(* CODESYS project proldPlcPrg.export

Project tree, tasks and I/O mapping:
  program PLC_PRG [LD]
*)

// PLC_PRG
PROGRAM PLC_PRG
VAR
	tmPusher1: TP;
	tmPusher2: TP;
	tmPusher3: TP;
END_VAR

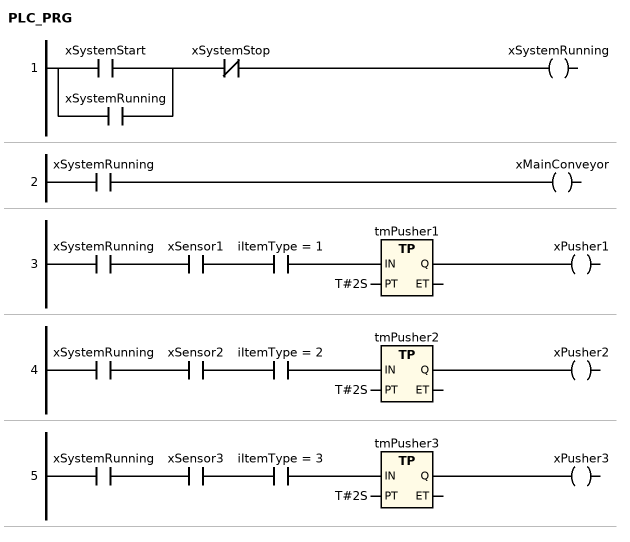
// NETWORK 1
xSystemRunning := (xSystemStart OR xSystemRunning) AND NOT xSystemStop;

// NETWORK 2
xMainConveyor := xSystemRunning;

// NETWORK 3
tmPusher1(IN := (xSystemRunning AND xSensor1) AND (iItemType = 1), PT := T#2S); // TP
xPusher1 := tmPusher1.Q;

// NETWORK 4
tmPusher2(IN := (xSystemRunning AND xSensor2) AND (iItemType = 2), PT := T#2S); // TP
xPusher2 := tmPusher2.Q;

// NETWORK 5
tmPusher3(IN := (xSystemRunning AND xSensor3) AND (iItemType = 3), PT := T#2S); // TP
xPusher3 := tmPusher3.Q;

END_PROGRAM
